FUNCTION_BLOCK TrackingLogic
VAR
	timerPistonInput: TOF;
	timerElapsedPistonInput: BOOL;
	counter: CTU;
	id: UDINT;
	item: Item;
	location: Location;
	timerTable: TOF;
	timerElapsedTable: BOOL;
	riseTrigTable: R_TRIG;
	riseTrigDetectedTable: BOOL;
	fallTrigTable: F_TRIG;
	fallTrigDetectedTable: BOOL;
	riseTrigPistonOutput: R_TRIG;
	riseTrigDetectedPistonOutput: BOOL;
	fallTrigBelt: F_TRIG;
	fallTrigDetectedBelt: bool;
	fallTrigPistonInput: F_TRIG;
	fallTrigDetectedPistonInput: BOOL;
END_VAR

//Piston Input logic
timerPistonInput(IN :=  NOT gvl.FotocellInput AND gvl.SwitchTablePosition, PT := T#1S, Q => timerElapsedPistonInput);
fallTrigPistonInput(CLK := gvl.PistonInputForward, Q => fallTrigDetectedPistonInput);
counter();
IF fallTrigDetectedPistonInput AND LocalVariables.Locations[2].Item.Id = 0 THEN
	LocalVariables.Locations[2].Item.Id := LocalVariables.Locations[1].Item.Id;
	LocalVariables.Locations[2].Item.Recipe := LocalVariables.Locations[1].Item.Recipe;
	LocalVariables.Locations[1].Item.Id := NULL;
ELSIF NOT gvl.FotocellInput THEN
	counter.CU := TRUE;
	id := counter.CV;
	LocalVariables.Locations[1].Item.Id := id;
	LocalVariables.Locations[1].Item.Recipe := LocalVariables.Recipe;
ELSE
	counter.CU := FALSE;
END_IF

//Table logic
riseTrigTable(CLK := gvl.SwitchPress, Q => riseTrigDetectedTable);
fallTrigTable(CLK:= gvl.SwitchPress, Q => fallTrigDetectedTable);
timerTable(IN := riseTrigDetectedTable, PT := LocalVariables.Recipe.WorkingTime, Q => timerElapsedTable);

IF riseTrigDetectedTable THEN
	LocalVariables.Locations[3].Item.Id := LocalVariables.Locations[2].Item.Id;
	LocalVariables.Locations[3].Item.Recipe := LocalVariables.Locations[2].Item.Recipe;
	LocalVariables.Locations[2].Item.Id := NULL;
	LocalVariables.Locations[2].Item.Recipe := LocalVariables.Recipe;
END_IF

IF fallTrigDetectedTable THEN
	LocalVariables.Locations[4].Item.Id := LocalVariables.Locations[3].Item.Id;
	LocalVariables.Locations[4].Item.Recipe := LocalVariables.Locations[3].Item.Recipe;
	LocalVariables.Locations[3].Item.Id := NULL;
	LocalVariables.Locations[3].Item.Recipe := LocalVariables.Recipe;
END_IF

//Piston Output logic
riseTrigPistonOutput(CLK := gvl.SwitchTableExit, Q => riseTrigDetectedPistonOutput);

IF riseTrigDetectedPistonOutput THEN
	LocalVariables.Locations[5].Item.Id := LocalVariables.Locations[4].Item.Id;
	LocalVariables.Locations[5].Item.Recipe := LocalVariables.Locations[4].Item.Recipe;
	LocalVariables.Locations[4].Item.Id := NULL;
	LocalVariables.Locations[4].Item.Recipe := LocalVariables.Recipe;
END_IF

//Belt logic
fallTrigBelt(CLK:= gvl.FotocellOutput, Q => fallTrigDetectedBelt);

IF gvl.FotocellOutput THEN
	LocalVariables.Locations[6].Item.Id := NULL;
	LocalVariables.Locations[6].Item.Recipe := LocalVariables.Recipe;
END_IF

IF fallTrigDetectedBelt THEN
	LocalVariables.Locations[6].Item.Id := LocalVariables.Locations[5].Item.Id;
	LocalVariables.Locations[6].Item.Recipe := LocalVariables.Locations[5].Item.Recipe;
	LocalVariables.Locations[5].Item.Id := NULL;
	LocalVariables.Locations[5].Item.Recipe := LocalVariables.Recipe;
END_IF

END_FUNCTION_BLOCK

(* stored: Version 1.1.0.1, ProductVersion 3.1.4024.12
   POU TrackingLogic: Id {8c28bcad-8b95-4b6d-89db-b0a98acfdd83}, SpecialFunc None *)
